(* CODESYS project WashingMachine (1).project

Project tree, tasks and I/O mapping:
  Device : CODESYS Control Win V3, 3S - Smart Software Solutions GmbH, version 3.5.15.10
    application Application
      libraries: Standard, * (System); VisuDialogs, * (System)
      task MainTask (cyclic, interval 100 ms, priority 1) calls Simulation_Program, GA_INSTANCES_prg, POLICY
      task VISU_TASK (cyclic, interval 100 ms, priority 31) calls VisuElems.Visu_Prg
      visualisation Visualization
      global variables GVL
      program Simulation_Program [ST]
      program BULLS_EYE_GA [SFC]: CHECK_DOOR_active, BUSY_active, LOCKING_DOOR_active, UNLOCKING_DOOR_active, END_active, END_exit, READY_active
      program TEMPERATURE_GA [SFC]: READY_active, BUSY_active, CHECK_TEMPERATURE_active, RESISTOR_ON_active, RESISTOR_OFF_active, CHECK_TEMPERATURE_exit
      program SOAP_GA [SFC]: CHECK_LEVEL_active, READY_active, BUSY_active, POURING_active, STOP_POURING_active, STOP_POURING_exit
      program WATER_GA [SFC]: READY_active, BUSY_active, FILLING_active, DRAINING_active, FILLING_exit, DRAINING_exit, END_active, END_exit, FAULT_OUT_DETECTOR_active, CHECK_LEVEL_active, FAULT_IN_DETECTOR_active
      program MOTOR_GA [SFC]: READY_active, BUSY_active, MOTOR_ON_active, MOTOR_OFF_active
      program POLICY [SFC]: RUN_PREWASH_exit, RUN_PREWASH_active, DOOR_UNLOCKED_active, CHECK_SOAP_active, RUN_PREWASH_NoRINSE_active, Init_exit, CHECK_DOOR_active, BULLS_EYE_LOCK_active, BULLS_EYE_LOCK_exit, RUN_WASH_active, RUN_WASH_exit, FINISHED_active, FAULT_MANAGER_active, Init_active, CHECK_TEMP_NUM_active, CHECK_PROG_NUM_active, BULLS_EYE_DOOR_UNLOCK_active, CHECK_STATE_active
      program PREWASH_WASH_POLICY [SFC]: Init_active, WATER_INTAKE_active, HEATING_active, FAULT_RESISTOR_active, EMPTYING_SOAP_active, MOTOR_ON_active, MOTOR_ON_exit, WATER_DRAIN_active, FAULT_OUT_VALVE_active, END_WASH_exit, END_WASH_active, HEATING_exit, EMPTYING_SOAP_exit, WATER_exit, RINSE_active, RINSE_exit, DUMMY_END_active, FAULT_HOT_DETECTOR_active, CHECK_FOR_STOP_active, WATER_DRAIN_entry
      program GA_INSTANCES_prg [FBD]
  text list GlobalTextList
*)

// Device/Application/GVL
{attribute 'qualified_only'}
VAR_GLOBAL
	temperature		: INT;		 	(*Sensor: current temperature of the water*)
	soaplevel		: INT; 			(*Sensor: current soap level*)
	waterlevel		: INT;			(*Sensor: current water level*)
	prog_number		: INT;			(*Input: program selected by the user*)
	temp_number		: INT; 			(*Input: temperature selected by the user*)
	run				: BOOL;			(*Input: if TRUE the washing machine works*)
	fillsoap		: BOOL; 		(*Input: if TRUE the soap tray is full*)
	bulls_eye_open	: BOOL := TRUE;	(*Input: if TRUE the door is open*)

	hot				: BOOL;			(*Actuator: if TRUE the resistor turns on*)
	motor_on		: BOOL;			(*Actuator: if TRUE the basket motor is turned on*)
	bulls_eye_lock	: BOOL;			(*Actuator: if TRUE the Door is locked*)
	emptysoap		: BOOL;			(*Actuator: if TRUE the soap tray is emptied*)
	fillwater		: BOOL;			(*Actuator: if TRUE the water is added*)
	emptywater		: BOOL;			(*Actuator: if TRUE the water is drained*)

	heat_alarm		: BOOL; 		(*Visualization: if TRUE alerts the user of the resistor fault*)
	water_in_alarm	: BOOL;			(*Visualization: if TRUE alerts the user of the water intake valve fault*)
	water_out_alarm	: BOOL; 		(*Visualization: if TRUE alerts the user of the water drain valve fault*)
	soap_alarm		: BOOL;			(*Visualization: if TRUE there is no soap*)
	prog_error		: BOOL;			(*Visualization: if TRUE the program selected is wrong*)
	temp_error		: BOOL;			(*Visualization: if TRUE the temperature selected is wrong*)
	rinse			: BOOL; 		(*Visualization: if TRUE the rinsing operation is going on*)
	prewash			: BOOL; 		(*Visualization: if TRUE the prewashing operation is going on*)
	wash			: BOOL; 		(*Visualization: if TRUE the washing operation is going on*)

	motor			: INT;			(*Only for simulation: angular position of the basket*)
	heat_fail		: BOOL;			(*Only for simulation: if TRUE the resistor cannot turn on*)
	water_in_fail	: BOOL;			(*Only for simulation: if TRUE the water intake valve is faulty*)
	water_out_fail	: BOOL;			(*Only for simulation: if TRUE the water drain valve is faulty*)
END_VAR

// Device/Application/Simulation_Program
PROGRAM Simulation_Program
VAR
		bulls_eye_open_past	:BOOL := TRUE;
END_VAR

(*Temperature value simulation*)
IF ((GVL.hot)AND(NOT GVL.heat_fail)) THEN 
	GVL.temperature := GVL.temperature + 1;
ELSE
	GVL.temperature := GVL.temperature - 1;
END_IF

IF GVL.temperature > 100 THEN 
	GVL.temperature := 100;
END_IF

IF GVL.temperature < 0 THEN 
	GVL.temperature := 0;
END_IF


(*Soap level simulation*)
IF GVL.fillsoap THEN 
	GVL.soaplevel := GVL.soaplevel + 5;
ELSIF GVL.emptysoap THEN 
	GVL.soaplevel := GVL.soaplevel - 3;
END_IF

IF GVL.soaplevel >= 50 THEN 
	GVL.soaplevel := 50;
	GVL.fillsoap := FALSE;
END_IF

IF GVL.soaplevel < 0 THEN 
	GVL.soaplevel := 0;
END_IF


(*Door state simulation*)
IF ((GVL.bulls_eye_open <> bulls_eye_open_past)AND(NOT GVL.bulls_eye_lock)) THEN 
	bulls_eye_open_past := GVL.bulls_eye_open ;
ELSIF GVL.bulls_eye_lock THEN
	GVL.bulls_eye_open := bulls_eye_open_past;
END_IF


(*Water level simulation*)
IF ((GVL.fillwater)AND(NOT GVL.water_in_fail)) THEN 
	GVL.waterlevel := GVL.waterlevel + 2;
ELSIF ((GVL.emptywater)AND(NOT GVL.water_out_fail)) THEN
	GVL.waterlevel := GVL.waterlevel - 4;
END_IF

IF GVL.waterlevel > 150 THEN 
	GVL.waterlevel := 150;
END_IF

IF GVL.waterlevel < 0 THEN 
	GVL.waterlevel := 0;
END_IF


(*Motor simulation*)
IF (GVL.motor_on) THEN 
	GVL.motor := GVL.motor + 10;
END_IF

IF GVL.motor > 360 THEN 
	GVL.motor := 0;
END_IF

END_PROGRAM

// Device/Application/GA_INSTANCES_prg
PROGRAM GA_INSTANCES_prg
VAR
END_VAR

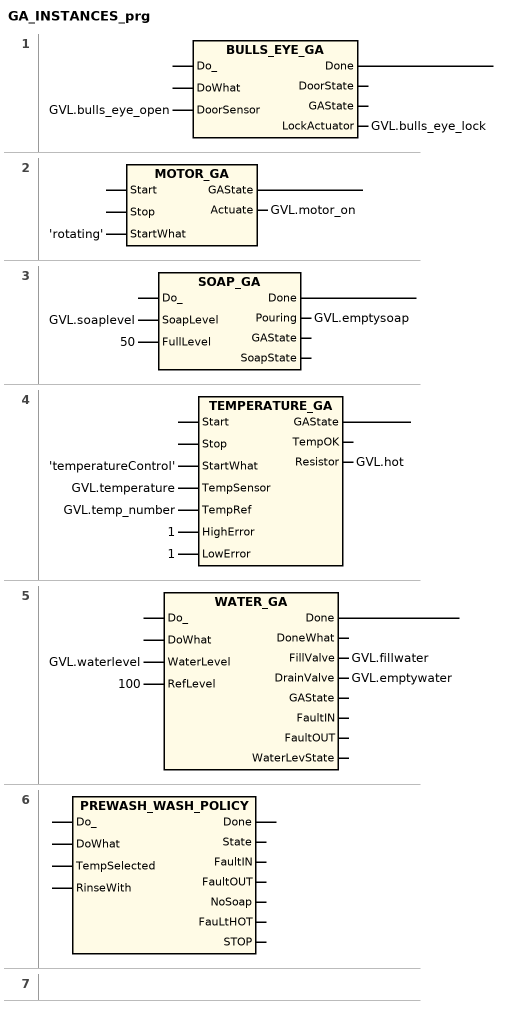
// NETWORK 1
BULLS_EYE_GA(DoorSensor := GVL.bulls_eye_open, LockActuator => GVL.bulls_eye_lock);

// NETWORK 2
MOTOR_GA(StartWhat := 'rotating', Actuate => GVL.motor_on);

// NETWORK 3
SOAP_GA(SoapLevel := GVL.soaplevel, FullLevel := 50, Pouring => GVL.emptysoap);

// NETWORK 4
TEMPERATURE_GA(StartWhat := 'temperatureControl', TempSensor := GVL.temperature, TempRef := GVL.temp_number, HighError := 1, LowError := 1, Resistor => GVL.hot);

// NETWORK 5
WATER_GA(WaterLevel := GVL.waterlevel, RefLevel := 100, FillValve => GVL.fillwater, DrainValve => GVL.emptywater);

// NETWORK 6
PREWASH_WASH_POLICY();

// NETWORK 7

END_PROGRAM

// Device/Application/BULLS_EYE_GA
PROGRAM BULLS_EYE_GA
//--------------------INPUT-----------------------
VAR_INPUT
	Do_:BOOL;
	DoWhat:STRING;
	DoorSensor:BOOL;
END_VAR
//-------------------OUTPUT-----------------------
VAR_OUTPUT
	Done:BOOL;
	DoorState:STRING;
	GAState:STRING;
	LockActuator:BOOL;
END_VAR
//--------------INTERNAL VARIABLES----------------
VAR
END_VAR

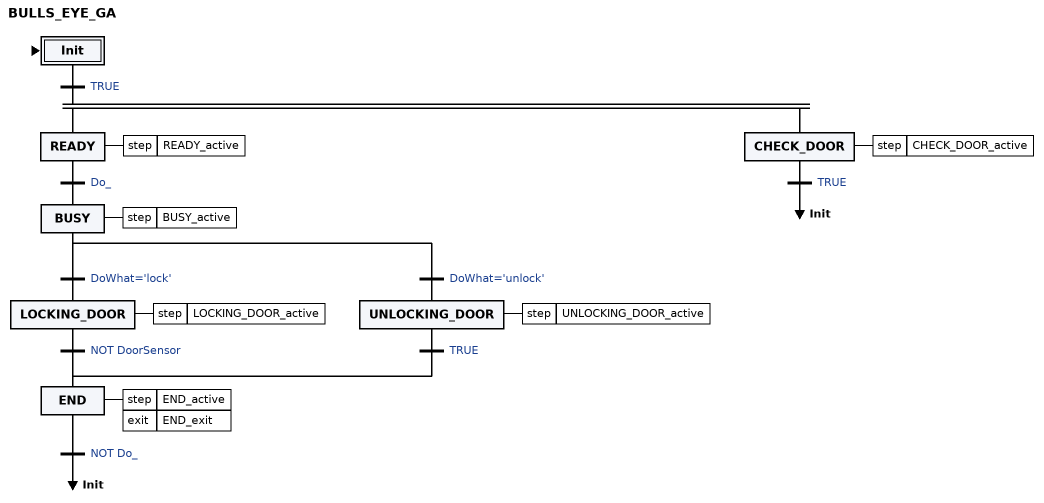
INITIAL_STEP Init:
END_STEP
TRANSITION FROM Init TO (READY, CHECK_DOOR)
    := TRUE;
END_TRANSITION
STEP READY:
    READY_active(N);  // step action
END_STEP
STEP CHECK_DOOR:
    CHECK_DOOR_active(N);  // step action
END_STEP
TRANSITION FROM CHECK_DOOR TO Init
    := TRUE;
END_TRANSITION
TRANSITION FROM READY TO BUSY
    := Do_;
END_TRANSITION
STEP BUSY:
    BUSY_active(N);  // step action
END_STEP
TRANSITION FROM BUSY TO LOCKING_DOOR
    := DoWhat='lock';
END_TRANSITION
STEP LOCKING_DOOR:
    LOCKING_DOOR_active(N);  // step action
END_STEP
TRANSITION FROM LOCKING_DOOR TO END
    := NOT DoorSensor;
END_TRANSITION
TRANSITION FROM BUSY TO UNLOCKING_DOOR
    := DoWhat='unlock';
END_TRANSITION
STEP UNLOCKING_DOOR:
    UNLOCKING_DOOR_active(N);  // step action
END_STEP
TRANSITION FROM UNLOCKING_DOOR TO END
    := TRUE;
END_TRANSITION
STEP END:
    END_active(N);  // step action
    END_exit(P0);  // exit action
END_STEP
TRANSITION FROM END TO Init
    := NOT Do_;
END_TRANSITION

ACTION CHECK_DOOR_active:
IF DoorSensor THEN
	DoorState:='open';
ELSE
	DoorState:='closed';
END_IF
END_ACTION

ACTION BUSY_active:
GAState:='busy';
END_ACTION

ACTION LOCKING_DOOR_active:
LockActuator:=TRUE;
END_ACTION

ACTION UNLOCKING_DOOR_active:
LockActuator:=FALSE;
END_ACTION

ACTION END_active:
Done:=TRUE;
END_ACTION

ACTION END_exit:
Done:=FALSE;
END_ACTION

ACTION READY_active:
GAState:='ready';
END_ACTION

END_PROGRAM

// Device/Application/MOTOR_GA
PROGRAM MOTOR_GA
//--------------------INPUT-----------------------
VAR_INPUT
	Start:BOOL;
	Stop:BOOL;
	StartWhat:STRING;
END_VAR
//-------------------OUTPUT-----------------------
VAR_OUTPUT
	GAState:STRING;
	Actuate:BOOL;
END_VAR
//--------------INTERNAL VARIABLES----------------
VAR
END_VAR

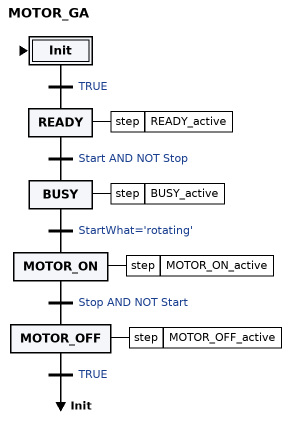
INITIAL_STEP Init:
END_STEP
TRANSITION FROM Init TO READY
    := TRUE;
END_TRANSITION
STEP READY:
    READY_active(N);  // step action
END_STEP
TRANSITION FROM READY TO BUSY
    := Start AND NOT Stop;
END_TRANSITION
STEP BUSY:
    BUSY_active(N);  // step action
END_STEP
TRANSITION FROM BUSY TO MOTOR_ON
    := StartWhat='rotating';
END_TRANSITION
STEP MOTOR_ON:
    MOTOR_ON_active(N);  // step action
END_STEP
TRANSITION FROM MOTOR_ON TO MOTOR_OFF
    := Stop AND NOT Start;
END_TRANSITION
STEP MOTOR_OFF:
    MOTOR_OFF_active(N);  // step action
END_STEP
TRANSITION FROM MOTOR_OFF TO Init
    := TRUE;
END_TRANSITION

ACTION READY_active:
GAState:='ready';
END_ACTION

ACTION BUSY_active:
GAState:='busy';
END_ACTION

ACTION MOTOR_ON_active:
Actuate:=TRUE;
END_ACTION

ACTION MOTOR_OFF_active:
Actuate:=FALSE;
END_ACTION

END_PROGRAM

// Device/Application/SOAP_GA
PROGRAM SOAP_GA
//--------------------INPUT-----------------------
VAR_INPUT
	Do_:BOOL;
	SoapLevel:INT;
	FullLevel:INT;
END_VAR
//-------------------OUTPUT-----------------------
VAR_OUTPUT
	Done:BOOL;
	Pouring:BOOL;
	GAState:STRING;
	SoapState:STRING;
END_VAR
//--------------INTERNAL VARIABLES----------------
VAR
	PouringTime:TIME := T#10S;
END_VAR

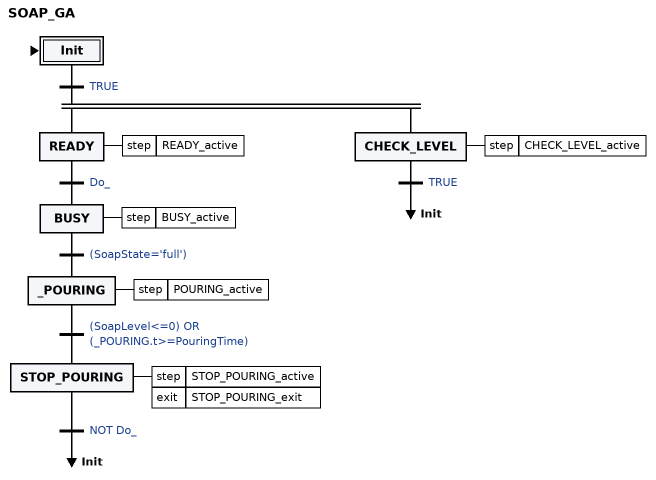
INITIAL_STEP Init:
END_STEP
TRANSITION FROM Init TO (READY, CHECK_LEVEL)
    := TRUE;
END_TRANSITION
STEP READY:
    READY_active(N);  // step action
END_STEP
STEP CHECK_LEVEL:
    CHECK_LEVEL_active(N);  // step action
END_STEP
TRANSITION FROM CHECK_LEVEL TO Init
    := TRUE;
END_TRANSITION
TRANSITION FROM READY TO BUSY
    := Do_;
END_TRANSITION
STEP BUSY:
    BUSY_active(N);  // step action
END_STEP
TRANSITION FROM BUSY TO _POURING
    := (SoapState='full');
END_TRANSITION
STEP _POURING:
    POURING_active(N);  // step action
END_STEP
TRANSITION FROM _POURING TO STOP_POURING
    := (SoapLevel<=0) OR (_POURING.t>=PouringTime);
END_TRANSITION
STEP STOP_POURING:
    STOP_POURING_active(N);  // step action
    STOP_POURING_exit(P0);  // exit action
END_STEP
TRANSITION FROM STOP_POURING TO Init
    := NOT Do_;
END_TRANSITION

ACTION CHECK_LEVEL_active:
IF SoapLevel>=FullLevel THEN
	SoapState:='full';
ELSE 
	SoapState:='notfull';	
END_IF
END_ACTION

ACTION READY_active:
GAState:='ready';
END_ACTION

ACTION BUSY_active:
GAState:='busy';
END_ACTION

ACTION POURING_active:
Pouring:=TRUE;
END_ACTION

ACTION STOP_POURING_active:
Pouring:=FALSE;
Done:=TRUE;
END_ACTION

ACTION STOP_POURING_exit:
Done:=FALSE;
END_ACTION

END_PROGRAM

// Device/Application/TEMPERATURE_GA
PROGRAM TEMPERATURE_GA
//--------------------INPUT-----------------------
VAR_INPUT
	Start:BOOL;
	Stop:BOOL;
	StartWhat:STRING;
	TempSensor:INT;
	TempRef:INT;
	HighError:INT;
	LowError:INT;
END_VAR
//-------------------OUTPUT-----------------------
VAR_OUTPUT
	GAState:STRING;
	TempOK:BOOL;
	Resistor:BOOL;
END_VAR
//--------------INTERNAL VARIABLES----------------
VAR
END_VAR

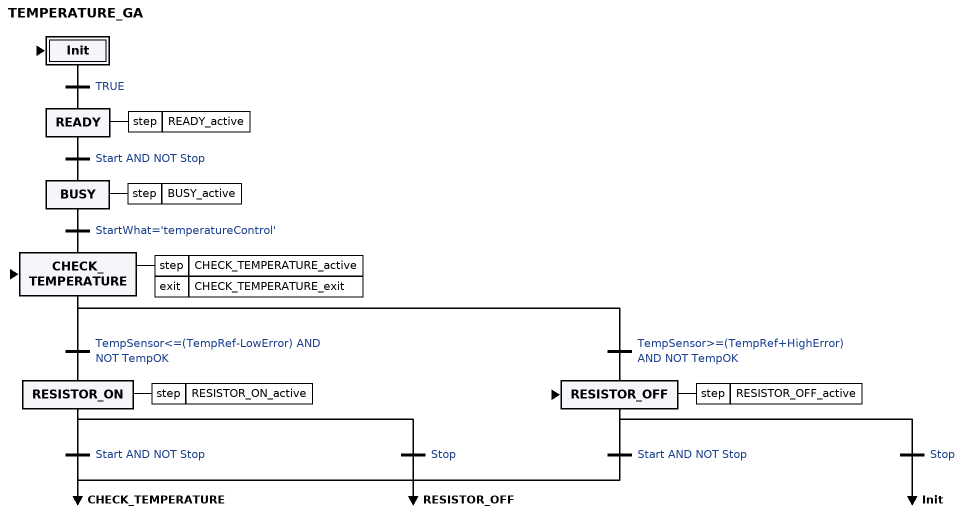
INITIAL_STEP Init:
END_STEP
TRANSITION FROM Init TO READY
    := TRUE;
END_TRANSITION
STEP READY:
    READY_active(N);  // step action
END_STEP
TRANSITION FROM READY TO BUSY
    := Start AND NOT Stop;
END_TRANSITION
STEP BUSY:
    BUSY_active(N);  // step action
END_STEP
TRANSITION FROM BUSY TO CHECK_TEMPERATURE
    := StartWhat='temperatureControl';
END_TRANSITION
STEP CHECK_TEMPERATURE:
    CHECK_TEMPERATURE_active(N);  // step action
    CHECK_TEMPERATURE_exit(P0);  // exit action
END_STEP
TRANSITION FROM CHECK_TEMPERATURE TO RESISTOR_ON
    := TempSensor<=(TempRef-LowError) AND NOT TempOK;
END_TRANSITION
STEP RESISTOR_ON:
    RESISTOR_ON_active(N);  // step action
END_STEP
TRANSITION FROM RESISTOR_ON TO CHECK_TEMPERATURE
    := Start AND NOT Stop;
END_TRANSITION
TRANSITION FROM RESISTOR_ON TO RESISTOR_OFF
    := Stop;
END_TRANSITION
TRANSITION FROM CHECK_TEMPERATURE TO RESISTOR_OFF
    := TempSensor>=(TempRef+HighError) AND NOT TempOK;
END_TRANSITION
STEP RESISTOR_OFF:
    RESISTOR_OFF_active(N);  // step action
END_STEP
TRANSITION FROM RESISTOR_OFF TO CHECK_TEMPERATURE
    := Start AND NOT Stop;
END_TRANSITION
TRANSITION FROM RESISTOR_OFF TO Init
    := Stop;
END_TRANSITION

ACTION READY_active:
GAState:='ready';
TempOK:=FALSE;
END_ACTION

ACTION BUSY_active:
GAState:='busy';
END_ACTION

ACTION CHECK_TEMPERATURE_active:
IF (TempSensor <= (TempRef + HighError)) AND (TempSensor >= (TempRef - LowError)) THEN
	TempOK:=TRUE;
ELSE
	TempOK:=FALSE;
END_IF
END_ACTION

ACTION RESISTOR_ON_active:
Resistor:=TRUE;
END_ACTION

ACTION RESISTOR_OFF_active:
Resistor:=FALSE;
END_ACTION

ACTION CHECK_TEMPERATURE_exit:
TempOK:=FALSE;
END_ACTION

END_PROGRAM

// Device/Application/WATER_GA
PROGRAM WATER_GA
//--------------------INPUT-----------------------
VAR_INPUT
	Do_:BOOL;
	DoWhat:STRING;
	WaterLevel:INT;
	RefLevel:INT;
END_VAR
//-------------------OUTPUT-----------------------
VAR_OUTPUT
	Done:BOOL;
	DoneWhat:STRING;
	FillValve:BOOL;
	DrainValve:BOOL;
	GAState:STRING;
	FaultIN:BOOL;
	FaultOUT:BOOL;
	WaterLevState:STRING;
END_VAR
//--------------INTERNAL VARIABLES----------------
VAR
	TimeFilling:TIME :=T#10S;
	TimeDraining:TIME :=T#10S;
    PrevLev:INT:=0;
	Count:INT:=0;
END_VAR

//WaterLevel>=RefLevel OR FILLING.t>TimeFilling
//WaterLevel<=0 OR DRAINING.t>TimeDraining

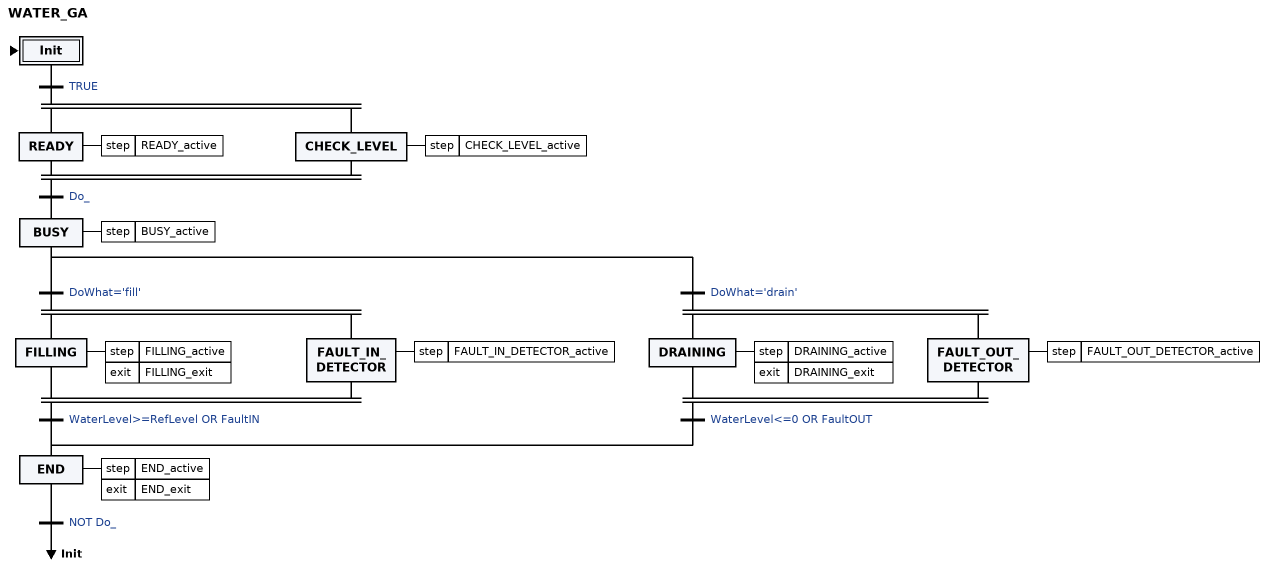
INITIAL_STEP Init:
END_STEP
TRANSITION FROM Init TO (READY, CHECK_LEVEL)
    := TRUE;
END_TRANSITION
STEP READY:
    READY_active(N);  // step action
END_STEP
STEP CHECK_LEVEL:
    CHECK_LEVEL_active(N);  // step action
END_STEP
TRANSITION FROM (READY, CHECK_LEVEL) TO BUSY
    := Do_;
END_TRANSITION
STEP BUSY:
    BUSY_active(N);  // step action
END_STEP
TRANSITION FROM BUSY TO (FILLING, FAULT_IN_DETECTOR)
    := DoWhat='fill';
END_TRANSITION
STEP FILLING:
    FILLING_active(N);  // step action
    FILLING_exit(P0);  // exit action
END_STEP
STEP FAULT_IN_DETECTOR:
    FAULT_IN_DETECTOR_active(N);  // step action
END_STEP
TRANSITION FROM (FILLING, FAULT_IN_DETECTOR) TO END
    := WaterLevel>=RefLevel OR FaultIN;
END_TRANSITION
TRANSITION FROM BUSY TO (DRAINING, FAULT_OUT_DETECTOR)
    := DoWhat='drain';
END_TRANSITION
STEP DRAINING:
    DRAINING_active(N);  // step action
    DRAINING_exit(P0);  // exit action
END_STEP
STEP FAULT_OUT_DETECTOR:
    FAULT_OUT_DETECTOR_active(N);  // step action
END_STEP
TRANSITION FROM (DRAINING, FAULT_OUT_DETECTOR) TO END
    := WaterLevel<=0 OR FaultOUT;
END_TRANSITION
STEP END:
    END_active(N);  // step action
    END_exit(P0);  // exit action
END_STEP
TRANSITION FROM END TO Init
    := NOT Do_;
END_TRANSITION

ACTION READY_active:
GAState:='ready';
END_ACTION

ACTION BUSY_active:
GAState:='busy';
END_ACTION

ACTION FILLING_active:
IF WaterLevel<RefLevel THEN
	WaterLevState:='notfull';	
	FillValve:=TRUE;
	DrainValve:=FALSE;
ELSE
WaterLevState:='full';	
END_IF
END_ACTION

ACTION DRAINING_active:
IF WaterLevel>0THEN
	WaterLevState:='full';	
	FillValve:=FALSE;
	DrainValve:=TRUE;
ELSE
	WaterLevState:='notfull';	
END_IF
END_ACTION

ACTION FILLING_exit:
FillValve:=FALSE;
DoneWhat:='fill';
END_ACTION

ACTION DRAINING_exit:
DrainValve:=FALSE;
DoneWhat:='drain';
END_ACTION

ACTION END_active:
Done:=TRUE;
PrevLev:=0;
END_ACTION

ACTION END_exit:
Done:=FALSE;
Count:=0;
END_ACTION

ACTION FAULT_OUT_DETECTOR_active:
//fault detection in the water_in_valve

FaultOUT:=FALSE;
IF Count=0THEN
	PrevLev:=WaterLevel;
END_IF
Count:=Count+1;
IF Count=20 THEN
	IF PrevLev <= WaterLevel THEN
		FaultOUT:=TRUE;
	ELSE
		FaultOUT:=FALSE;
	END_IF
	Count:=0;
END_IF
END_ACTION

ACTION CHECK_LEVEL_active:
IF WaterLevel>=RefLevel THEN
	WaterLevState:='full';
ELSE 
	WaterLevState:='notfull';	
END_IF

FaultIN:=FALSE;
FaultOUT:=FALSE;
END_ACTION

ACTION FAULT_IN_DETECTOR_active:
//fault detection in the water_in_valve

FaultIN:=FALSE;
Count:=Count+1;
IF Count=20 THEN
	IF PrevLev >= WaterLevel THEN
		FaultIN:=TRUE;
	ELSE
		FaultIN:=FALSE;
	END_IF
	PrevLev:=WaterLevel;
	Count:=0;
END_IF
END_ACTION

END_PROGRAM

// Device/Application/PREWASH_WASH_POLICY
PROGRAM PREWASH_WASH_POLICY
//--------------------INPUT-----------------------
VAR_INPUT
	Do_:BOOL;
	DoWhat:STRING;
	TempSelected:INT;
	RinseWith:BOOL;
END_VAR
//-------------------OUTPUT-----------------------
VAR_OUTPUT
	Done:BOOL;
	State:STRING;
	FaultIN:BOOL;
	FaultOUT:BOOL;
	NoSoap:BOOL;
	FauLtHOT:BOOL;
	STOP:BOOL;
END_VAR
//--------------INTERNAL VARIABLES----------------
VAR
	OK:BOOL;
	HeatingMaxTime:TIME:=T#10S;
	SoapOK:BOOL;
	Count:INT:=0;
	PrevTemp:INT:=0;
END_VAR

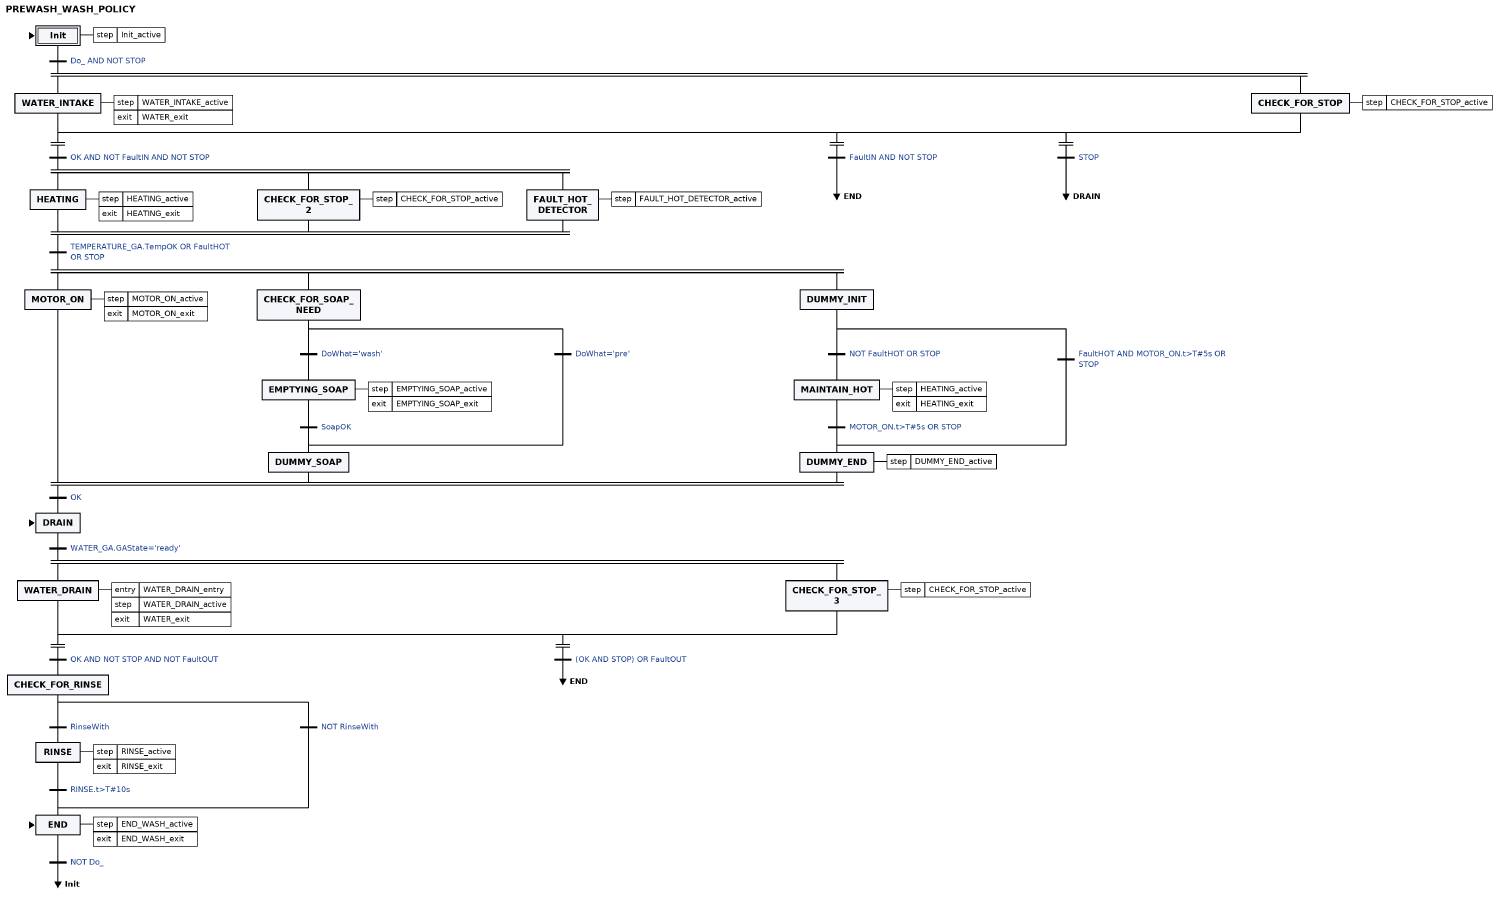
INITIAL_STEP Init:
    Init_active(N);  // step action
END_STEP
TRANSITION FROM Init TO (WATER_INTAKE, CHECK_FOR_STOP)
    := Do_ AND NOT STOP;
END_TRANSITION
STEP WATER_INTAKE:
    WATER_INTAKE_active(N);  // step action
    WATER_exit(P0);  // exit action
END_STEP
STEP CHECK_FOR_STOP:
    CHECK_FOR_STOP_active(N);  // step action
END_STEP
TRANSITION FROM (WATER_INTAKE, CHECK_FOR_STOP) TO (HEATING, CHECK_FOR_STOP_2, FAULT_HOT_DETECTOR)
    := OK AND NOT FaultIN AND NOT STOP;
END_TRANSITION
TRANSITION FROM (WATER_INTAKE, CHECK_FOR_STOP) TO END
    := FaultIN AND NOT STOP;
END_TRANSITION
TRANSITION FROM (WATER_INTAKE, CHECK_FOR_STOP) TO DRAIN
    := STOP;
END_TRANSITION
STEP HEATING:
    HEATING_active(N);  // step action
    HEATING_exit(P0);  // exit action
END_STEP
STEP CHECK_FOR_STOP_2:
    CHECK_FOR_STOP_active(N);  // step action
END_STEP
STEP FAULT_HOT_DETECTOR:
    FAULT_HOT_DETECTOR_active(N);  // step action
END_STEP
TRANSITION FROM (HEATING, CHECK_FOR_STOP_2, FAULT_HOT_DETECTOR) TO (MOTOR_ON, CHECK_FOR_SOAP_NEED, DUMMY_INIT)
    := TEMPERATURE_GA.TempOK OR FaultHOT OR STOP;
END_TRANSITION
STEP MOTOR_ON:
    MOTOR_ON_active(N);  // step action
    MOTOR_ON_exit(P0);  // exit action
END_STEP
STEP CHECK_FOR_SOAP_NEED:
END_STEP
TRANSITION FROM CHECK_FOR_SOAP_NEED TO EMPTYING_SOAP
    := DoWhat='wash';
END_TRANSITION
STEP EMPTYING_SOAP:
    EMPTYING_SOAP_active(N);  // step action
    EMPTYING_SOAP_exit(P0);  // exit action
END_STEP
TRANSITION FROM EMPTYING_SOAP TO DUMMY_SOAP
    := SoapOK;
END_TRANSITION
TRANSITION FROM CHECK_FOR_SOAP_NEED TO DUMMY_SOAP
    := DoWhat='pre';
END_TRANSITION
STEP DUMMY_SOAP:
END_STEP
STEP DUMMY_INIT:
END_STEP
TRANSITION FROM DUMMY_INIT TO MAINTAIN_HOT
    := NOT FaultHOT OR STOP;
END_TRANSITION
STEP MAINTAIN_HOT:
    HEATING_active(N);  // step action
    HEATING_exit(P0);  // exit action
END_STEP
TRANSITION FROM MAINTAIN_HOT TO DUMMY_END
    := MOTOR_ON.t>T#5s OR STOP;
END_TRANSITION
TRANSITION FROM DUMMY_INIT TO DUMMY_END
    := FaultHOT AND MOTOR_ON.t>T#5s OR STOP;
END_TRANSITION
STEP DUMMY_END:
    DUMMY_END_active(N);  // step action
END_STEP
TRANSITION FROM (MOTOR_ON, DUMMY_SOAP, DUMMY_END) TO DRAIN
    := OK;
END_TRANSITION
STEP DRAIN:
END_STEP
TRANSITION FROM DRAIN TO (WATER_DRAIN, CHECK_FOR_STOP_3)
    := WATER_GA.GAState='ready';
END_TRANSITION
STEP WATER_DRAIN:
    WATER_DRAIN_entry(P1);  // entry action
    WATER_DRAIN_active(N);  // step action
    WATER_exit(P0);  // exit action
END_STEP
STEP CHECK_FOR_STOP_3:
    CHECK_FOR_STOP_active(N);  // step action
END_STEP
TRANSITION FROM (WATER_DRAIN, CHECK_FOR_STOP_3) TO CHECK_FOR_RINSE
    := OK AND NOT STOP AND NOT FaultOUT;
END_TRANSITION
TRANSITION FROM (WATER_DRAIN, CHECK_FOR_STOP_3) TO END
    := (OK AND STOP) OR FaultOUT;
END_TRANSITION
STEP CHECK_FOR_RINSE:
END_STEP
TRANSITION FROM CHECK_FOR_RINSE TO RINSE
    := RinseWith;
END_TRANSITION
STEP RINSE:
    RINSE_active(N);  // step action
    RINSE_exit(P0);  // exit action
END_STEP
TRANSITION FROM RINSE TO END
    := RINSE.t>T#10s;
END_TRANSITION
TRANSITION FROM CHECK_FOR_RINSE TO END
    := NOT RinseWith;
END_TRANSITION
STEP END:
    END_WASH_active(N);  // step action
    END_WASH_exit(P0);  // exit action
END_STEP
TRANSITION FROM END TO Init
    := NOT Do_;
END_TRANSITION

ACTION Init_active:
State:='init';
FaultIN:=FALSE;
FaultOUT:=FALSE;
NoSoap:=FALSE;
FauLtHOT:=FALSE;
IF GVL.run THEN
	STOP:=FALSE;
ELSE
	STOP:=TRUE;
END_IF
END_ACTION

ACTION WATER_INTAKE_active:
FaultIN:=FALSE;
IF WATER_GA.WaterLevState='notfull' THEN

		IF WATER_GA.GAState='ready' THEN
			WATER_GA.Do_:=TRUE;
			WATER_GA.DoWhat:='fill';
		END_IF

		IF WATER_GA.Done AND WATER_GA.GAState='busy' THEN
			FaultIN:=WATER_GA.FaultIN;
			OK:=TRUE;
		END_IF
		
	ELSE
		OK:=TRUE;
END_IF	
IF NOT(State='fault') THEN
	State:=DoWhat;
END_IF
END_ACTION

ACTION HEATING_active:
FaultHOT:=FALSE;
IF TEMPERATURE_GA.GAState= 'ready' THEN
		TEMPERATURE_GA.Start:=TRUE;
		TEMPERATURE_GA.Stop:=FALSE;
END_IF
END_ACTION

ACTION FAULT_RESISTOR_active:
FaultHOT:=TRUE;
State:='fault';
END_ACTION

ACTION EMPTYING_SOAP_active:
NoSoap:=FALSE;
IF SOAP_GA.SoapState='full' THEN
	NoSoap:=FALSE;
ELSE
	NoSoap:=TRUE;
END_IF

IF SOAP_GA.SoapLevel>0 THEN
	IF SOAP_GA.GAState='ready'THEN
		SOAP_GA.Do_:=TRUE;
	END_IF
	IF SOAP_GA.Done AND SOAP_GA.GAState='busy' THEN
		SOAP_GA.Do_:=FALSE;
		SoapOK:=SOAP_GA.Done;
	END_IF
ELSE
	SoapOK:=TRUE;
END_IF
END_ACTION

ACTION MOTOR_ON_active:
IF MOTOR_GA.GAState= 'ready' THEN
		MOTOR_GA.Start:=TRUE;
		MOTOR_GA.Stop:=FALSE;
END_IF
END_ACTION

ACTION MOTOR_ON_exit:
IF MOTOR_GA.GAState= 'busy' THEN
		MOTOR_GA.Start:=FALSE;
		MOTOR_GA.Stop:=TRUE;
END_IF
END_ACTION

ACTION WATER_DRAIN_active:
FaultOUT:=FALSE;
IF WATER_GA.WaterLevState='full'THEN
		
		IF WATER_GA.GAState='ready' THEN
			WATER_GA.Do_:=TRUE;
			WATER_GA.DoWhat:='drain';
		END_IF

		IF WATER_GA.Done AND WATER_GA.GAState='busy' THEN
			FaultOUT:=WATER_GA.FaultOUT;
			OK:=TRUE;
		END_IF
		
	ELSE
		OK:=TRUE;
END_IF
END_ACTION

ACTION FAULT_OUT_VALVE_active:
GVL.water_out_alarm:=TRUE;
FaultOUT:=TRUE;
END_ACTION

ACTION END_WASH_exit:
Done:=FALSE;
State:='init';
STOP:=FALSE;
END_ACTION

ACTION END_WASH_active:
IF ((NOT FaultIN) AND (NOT FaultOUT) AND (NOT FaultHOT))THEN
	State:='end';
ELSE
	State:='fault';
END_IF

IF GVL.run THEN
	STOP:=FALSE;
ELSE
	STOP:=TRUE;
END_IF

Done:=TRUE;
Count:=0;
PrevTemp:=0;
END_ACTION

ACTION HEATING_exit:
IF TEMPERATURE_GA.GAState= 'busy' THEN
		TEMPERATURE_GA.Start:=FALSE;
		TEMPERATURE_GA.Stop:=TRUE;
END_IF
Count:=0;
STOP:=FALSE;
END_ACTION

ACTION EMPTYING_SOAP_exit:
SoapOK:=FALSE;
END_ACTION

ACTION WATER_exit:
OK:=FALSE;
WATER_GA.Do_:=FALSE;
STOP:=FALSE;
END_ACTION

ACTION RINSE_active:
IF MOTOR_GA.GAState= 'ready' THEN
		MOTOR_GA.Start:=TRUE;
		MOTOR_GA.Stop:=FALSE;
END_IF
IF NOT(State='fault') THEN
	State:='rinse';
END_IF
END_ACTION

ACTION RINSE_exit:
IF MOTOR_GA.GAState= 'busy' THEN
		MOTOR_GA.Start:=FALSE;
		MOTOR_GA.Stop:=TRUE;
END_IF
END_ACTION

ACTION DUMMY_END_active:
OK:=TRUE;
END_ACTION

ACTION FAULT_HOT_DETECTOR_active:
FaultHOT:=FALSE;
Count:=Count+1;
IF Count=20 THEN
	IF PrevTemp >= TEMPERATURE_GA.TempSensor THEN
		FaultHOT:=TRUE;
		State:='fault';
	ELSE
		FaultHOT:=FALSE;
	END_IF
	PrevTemp:=TEMPERATURE_GA.TempSensor;
	Count:=0;
END_IF
END_ACTION

ACTION CHECK_FOR_STOP_active:
IF GVL.run THEN
	STOP:=FALSE;
ELSE
	STOP:=TRUE;
END_IF
END_ACTION

ACTION WATER_DRAIN_entry:
OK:=FALSE;
END_ACTION

END_PROGRAM

// Device/Application/POLICY
PROGRAM POLICY
VAR
	TempNumOK:BOOL;
	ProgNumOK:BOOL;
	RunOK:BOOL;
	WashOK:BOOL;
	STOP:BOOL;
	DoorOK:BOOL;
	TempOK:BOOL;


END_VAR

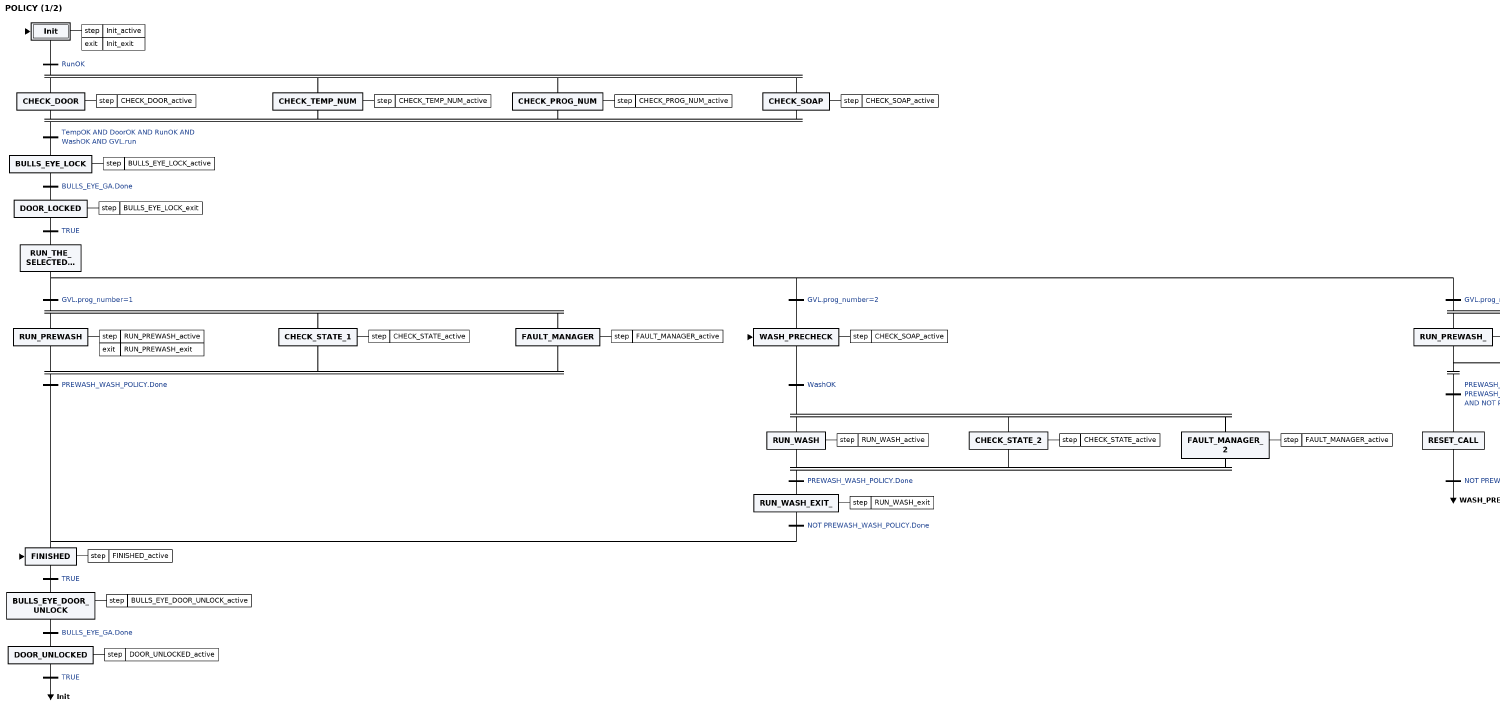
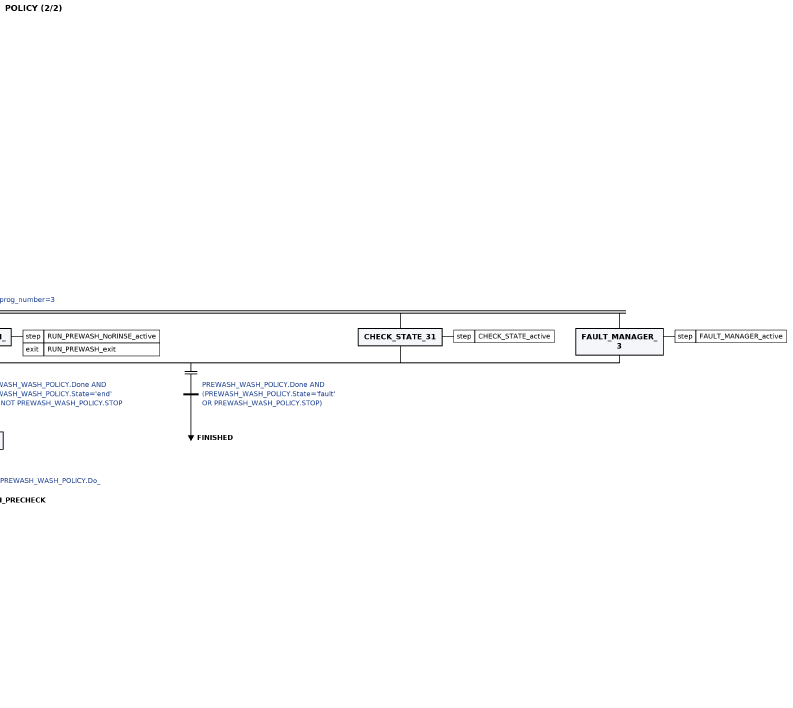
INITIAL_STEP Init:
    Init_active(N);  // step action
    Init_exit(P0);  // exit action
END_STEP
TRANSITION FROM Init TO (CHECK_DOOR, CHECK_TEMP_NUM, CHECK_PROG_NUM, CHECK_SOAP)
    := RunOK;
END_TRANSITION
STEP CHECK_DOOR:
    CHECK_DOOR_active(N);  // step action
END_STEP
STEP CHECK_TEMP_NUM:
    CHECK_TEMP_NUM_active(N);  // step action
END_STEP
STEP CHECK_PROG_NUM:
    CHECK_PROG_NUM_active(N);  // step action
END_STEP
STEP CHECK_SOAP:
    CHECK_SOAP_active(N);  // step action
END_STEP
TRANSITION FROM (CHECK_DOOR, CHECK_TEMP_NUM, CHECK_PROG_NUM, CHECK_SOAP) TO BULLS_EYE_LOCK
    := TempOK AND DoorOK AND RunOK AND WashOK AND GVL.run;
END_TRANSITION
STEP BULLS_EYE_LOCK:
    BULLS_EYE_LOCK_active(N);  // step action
END_STEP
TRANSITION FROM BULLS_EYE_LOCK TO DOOR_LOCKED
    := BULLS_EYE_GA.Done;
END_TRANSITION
STEP DOOR_LOCKED:
    BULLS_EYE_LOCK_exit(N);  // step action
END_STEP
TRANSITION FROM DOOR_LOCKED TO RUN_THE_SELECTED_PROGRAM
    := TRUE;
END_TRANSITION
STEP RUN_THE_SELECTED_PROGRAM:
END_STEP
TRANSITION FROM RUN_THE_SELECTED_PROGRAM TO (RUN_PREWASH, CHECK_STATE_1, FAULT_MANAGER)
    := GVL.prog_number=1;
END_TRANSITION
STEP RUN_PREWASH:
    RUN_PREWASH_active(N);  // step action
    RUN_PREWASH_exit(P0);  // exit action
END_STEP
STEP CHECK_STATE_1:
    CHECK_STATE_active(N);  // step action
END_STEP
STEP FAULT_MANAGER:
    FAULT_MANAGER_active(N);  // step action
END_STEP
TRANSITION FROM (RUN_PREWASH, CHECK_STATE_1, FAULT_MANAGER) TO FINISHED
    := PREWASH_WASH_POLICY.Done;
END_TRANSITION
TRANSITION FROM RUN_THE_SELECTED_PROGRAM TO WASH_PRECHECK
    := GVL.prog_number=2;
END_TRANSITION
STEP WASH_PRECHECK:
    CHECK_SOAP_active(N);  // step action
END_STEP
TRANSITION FROM WASH_PRECHECK TO (RUN_WASH, CHECK_STATE_2, FAULT_MANAGER_2)
    := WashOK;
END_TRANSITION
STEP RUN_WASH:
    RUN_WASH_active(N);  // step action
END_STEP
STEP CHECK_STATE_2:
    CHECK_STATE_active(N);  // step action
END_STEP
STEP FAULT_MANAGER_2:
    FAULT_MANAGER_active(N);  // step action
END_STEP
TRANSITION FROM (RUN_WASH, CHECK_STATE_2, FAULT_MANAGER_2) TO RUN_WASH_EXIT_
    := PREWASH_WASH_POLICY.Done;
END_TRANSITION
STEP RUN_WASH_EXIT_:
    RUN_WASH_exit(N);  // step action
END_STEP
TRANSITION FROM RUN_WASH_EXIT_ TO FINISHED
    := NOT PREWASH_WASH_POLICY.Done;
END_TRANSITION
TRANSITION FROM RUN_THE_SELECTED_PROGRAM TO (RUN_PREWASH_, CHECK_STATE_31, FAULT_MANAGER_3)
    := GVL.prog_number=3;
END_TRANSITION
STEP RUN_PREWASH_:
    RUN_PREWASH_NoRINSE_active(N);  // step action
    RUN_PREWASH_exit(P0);  // exit action
END_STEP
STEP CHECK_STATE_31:
    CHECK_STATE_active(N);  // step action
END_STEP
STEP FAULT_MANAGER_3:
    FAULT_MANAGER_active(N);  // step action
END_STEP
TRANSITION FROM (RUN_PREWASH_, CHECK_STATE_31, FAULT_MANAGER_3) TO RESET_CALL
    := PREWASH_WASH_POLICY.Done AND PREWASH_WASH_POLICY.State='end' AND NOT PREWASH_WASH_POLICY.STOP;
END_TRANSITION
STEP RESET_CALL:
END_STEP
TRANSITION FROM RESET_CALL TO WASH_PRECHECK
    := NOT PREWASH_WASH_POLICY.Do_;
END_TRANSITION
TRANSITION FROM (RUN_PREWASH_, CHECK_STATE_31, FAULT_MANAGER_3) TO FINISHED
    := PREWASH_WASH_POLICY.Done AND (PREWASH_WASH_POLICY.State='fault' OR PREWASH_WASH_POLICY.STOP);
END_TRANSITION
STEP FINISHED:
    FINISHED_active(N);  // step action
END_STEP
TRANSITION FROM FINISHED TO BULLS_EYE_DOOR_UNLOCK
    := TRUE;
END_TRANSITION
STEP BULLS_EYE_DOOR_UNLOCK:
    BULLS_EYE_DOOR_UNLOCK_active(N);  // step action
END_STEP
TRANSITION FROM BULLS_EYE_DOOR_UNLOCK TO DOOR_UNLOCKED
    := BULLS_EYE_GA.Done;
END_TRANSITION
STEP DOOR_UNLOCKED:
    DOOR_UNLOCKED_active(N);  // step action
END_STEP
TRANSITION FROM DOOR_UNLOCKED TO Init
    := TRUE;
END_TRANSITION

ACTION RUN_PREWASH_exit:
PREWASH_WASH_POLICY.Do_:=FALSE;
END_ACTION

ACTION RUN_PREWASH_active:
PREWASH_WASH_POLICY.Do_:=TRUE;
PREWASH_WASH_POLICY.DoWhat:='pre';
PREWASH_WASH_POLICY.RinseWith:=TRUE;
END_ACTION

ACTION DOOR_UNLOCKED_active:
IF BULLS_EYE_GA.GAState='busy' THEN
	BULLS_EYE_GA.Do_:=FALSE;
END_IF
END_ACTION

ACTION CHECK_SOAP_active:
IF (SOAP_GA.SoapState='full')OR(GVL.prog_number=1)THEN
	WashOK:=TRUE;
	GVL.soap_alarm:=FALSE;
ELSE
	WashOK:=FALSE;
	GVL.soap_alarm:=TRUE;
END_IF
END_ACTION

ACTION RUN_PREWASH_NoRINSE_active:
PREWASH_WASH_POLICY.Do_:=TRUE;
PREWASH_WASH_POLICY.DoWhat:='pre';
PREWASH_WASH_POLICY.RinseWith:=FALSE;
END_ACTION

ACTION Init_exit:
RunOK:=FALSE;
END_ACTION

ACTION CHECK_DOOR_active:
IF BULLS_EYE_GA.DoorState='open'THEN
	DoorOK:=FALSE;
END_IF

IF BULLS_EYE_GA.DoorState='closed' THEN
	DoorOK:=TRUE;
END_IF
END_ACTION

ACTION BULLS_EYE_LOCK_active:
IF BULLS_EYE_GA.GAState='ready' THEN
	BULLS_EYE_GA.Do_:=TRUE;
	BULLS_EYE_GA.DoWhat:='lock';
END_IF
END_ACTION

ACTION BULLS_EYE_LOCK_exit:
IF BULLS_EYE_GA.GAState='busy' THEN
	BULLS_EYE_GA.Do_:=FALSE;
END_IF
END_ACTION

ACTION RUN_WASH_active:
PREWASH_WASH_POLICY.Do_:=TRUE;
PREWASH_WASH_POLICY.DoWhat:='wash';
PREWASH_WASH_POLICY.RinseWith:=TRUE;
END_ACTION

ACTION RUN_WASH_exit:
PREWASH_WASH_POLICY.Do_:=FALSE;
END_ACTION

ACTION FINISHED_active:
GVL.run:=FALSE;
END_ACTION

ACTION FAULT_MANAGER_active:
IF PREWASH_WASH_POLICY.FaultIN THEN
	GVL.water_in_alarm:=TRUE;
ELSE
	GVL.water_in_alarm:=STOP:=FALSE;
END_IF
IF PREWASH_WASH_POLICY.FaultOUT THEN
	GVL.water_out_alarm:=TRUE;
ELSE
	GVL.water_OUT_alarm:=STOP:=FALSE;
END_IF
IF PREWASH_WASH_POLICY.FaultHOT THEN
	GVL.heat_alarm:=TRUE;
ELSE
	GVL.heat_alarm:=FALSE;
END_IF
IF PREWASH_WASH_POLICY.NoSoap THEN
	GVL.soap_alarm:=TRUE;
	WashOK:=FALSE;
ELSE
	GVL.soap_alarm:=FALSE;
	WashOK:=TRUE;
END_IF
END_ACTION

ACTION Init_active:
IF GVL.water_in_alarm OR GVL.water_out_alarm THEN
	RunOK:=FALSE;
ELSE
	RunOK:=TRUE;
END_IF
END_ACTION

ACTION CHECK_TEMP_NUM_active:
IF (GVL.temp_number=30)OR(GVL.temp_number=60)OR(GVL.temp_number=90)THEN
	TempOK:=TRUE;
	GVL.temp_error:=FALSE;
ELSE
	TempOK:=FALSE;
	GVL.temp_error:=TRUE;
END_IF
END_ACTION

ACTION CHECK_PROG_NUM_active:
IF (GVL.prog_number=1) OR (GVL.prog_number=2) OR (GVL.prog_number=3) THEN
	RunOK:=TRUE;
	GVL.prog_error:=FALSE;
ELSE
	RunOK:=FALSE;
	GVL.prog_error:=TRUE;
END_IF
END_ACTION

ACTION BULLS_EYE_DOOR_UNLOCK_active:
IF BULLS_EYE_GA.GAState='ready' THEN
	BULLS_EYE_GA.Do_:=TRUE;
	BULLS_EYE_GA.DoWhat:='unlock';
END_IF
END_ACTION

ACTION CHECK_STATE_active:
IF (PREWASH_WASH_POLICY.State='pre') THEN
	GVL.prewash:=TRUE;
	GVL.wash:=FALSE;
	GVL.rinse:=FALSE;
END_IF

IF (PREWASH_WASH_POLICY.State='rinse') THEN
	GVL.prewash:=FALSE;
	GVL.wash:=FALSE;
	GVL.rinse:=TRUE;
END_IF

IF (PREWASH_WASH_POLICY.State='wash') THEN
	GVL.prewash:=FALSE;
	GVL.wash:=TRUE;
	GVL.rinse:=FALSE;
END_IF

IF PREWASH_WASH_POLICY.State='fault' OR PREWASH_WASH_POLICY.State='end' THEN
	GVL.prewash:=FALSE;
	GVL.wash:=FALSE;
	GVL.rinse:=FALSE;
END_IF
END_ACTION

END_PROGRAM

// Device/Application/Visualization
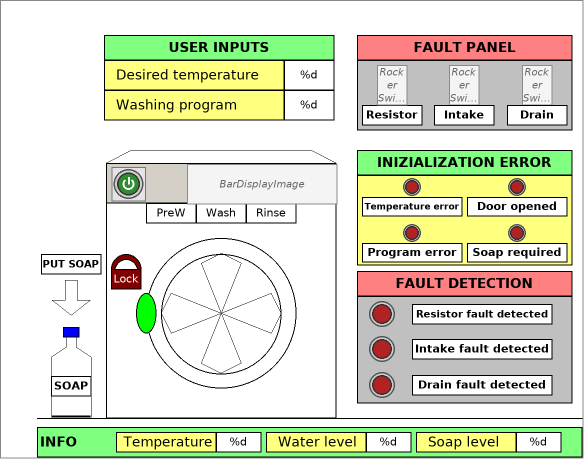
VISUALIZATION Visualization  // 584x459
    Line (37,418) (582,418)
    Rectangle (106,178 230x240)
    Ellipse (162,254 118x118)
    Rectangle (161,255 120x120)
        p1126004900: -GVL.waterlevel/3*2
    Ellipse (146,238 150x150)
    Ellipse (161,254 120x120)
    Polygon (221,253) (201,263) (221,313) (171,293) (161,313) (171,333) (221,313) (201,363) (221,373) (241,363) (221,313) (271,333) (281,313) (271,293) (221,313) (241,263)
        p2858320360: GVL.motor
    Ellipse (136,293 20x40), colour toggle: GVL.bulls_eye_open
        toggle GVL.bulls_eye_open
    Ellipse (111,254 30x30), colour toggle: GVL.bulls_eye_lock
    Ellipse (114,259 24x27)
    Rectangle (111,269 30x20), "Lock", colour toggle: GVL.bulls_eye_lock
    Rectangle (106,163 230x40)
    Rectangle (146,203 50x20), "PreW", colour toggle: GVL.prewash
    Rectangle (196,203 50x20), "Wash", colour toggle: GVL.wash
    Rectangle (246,203 50x20), "Rinse", colour toggle: GVL.rinse
    Polygon (106,163) (131,150) (311,150) (336,163)
    PowerSwitch (111,167 35x34), variable: GVL.run, behaviour: TOGGLE, style: Switch-PowerSwitch-Green
    BarDisplayImage (187,164 150x40), value: GVL.temperature, style: BarDisplayImage-Gray, scale format: %.0f, scale 0..90
    Polygon (51,417) (51,357) (66,347) (66,332) (76,332) (76,347) (91,357) (91,417)
    Rectangle (63,327 16x10)
    Rectangle (104,60 180x30), "Desired temperature"
        OnMouseDown: write GVL.temp_number via VisuDialogs.Numpad, min 0, max 100, format 0
    Rectangle (104,90 180x30), "Washing program"
        OnMouseDown: write GVL.prog_number via VisuDialogs.Numpad, min 0, max 100, format 0
    Rectangle (104,35 230x25), "USER INPUTS"
    Rectangle (284,60 50x30), "%d", text variable: GVL.temp_number
    Rectangle (284,90 50x30), "%d", text variable: GVL.prog_number
    Rectangle (37,427 545x30), "INFO"
    Rectangle (116,432 100x20), "Temperature"
    Rectangle (357,150 215x25), "INIZIALIZATION ERROR"
    Rectangle (216,432 45x20), "%d", text variable: GVL.temperature
    Rectangle (266,432 100x20), "Water level"
    Rectangle (366,432 45x20), "%d", text variable: GVL.waterlevel
    Rectangle (416,432 100x20), "Soap level"
    Rectangle (516,432 45x20), "%d", text variable: GVL.soaplevel
    Rectangle (357,175 215x90)
    Lamp1 (402,177 20x20), variable: GVL.temp_error, style: Lamp-Lamp1-Red
    Rectangle (362,197 100x19), "Temperature error"
    Lamp1 (507,177 20x20), variable: GVL.bulls_eye_open, style: Lamp-Lamp1-Red
    Rectangle (467,197 100x19), "Door opened"
    Lamp1 (402,223 20x20), variable: GVL.prog_error, style: Lamp-Lamp1-Red
    Rectangle (362,243 100x19), "Program error"
    Lamp1 (507,223 20x20), variable: GVL.soap_alarm, style: Lamp-Lamp1-Red
    Rectangle (467,243 100x19), "Soap required"
    Rectangle (357,35 215x25), "FAULT PANEL"
    Rectangle (357,60 215x70)
    Rectangle (362,105 60x20), "Resistor"
    RockerSwitch (377,65 30x40), variable: GVL.heat_fail, behaviour: TOGGLE, style: Switch-RockerSwitch-Red
    RockerSwitch (449,65 30x40), variable: GVL.water_in_fail, behaviour: TOGGLE, style: Switch-RockerSwitch-Red
    Rectangle (434,105 60x20), "Intake"
    RockerSwitch (522,65 30x40), variable: GVL.water_out_fail, behaviour: TOGGLE, style: Switch-RockerSwitch-Red
    Rectangle (507,105 60x20), "Drain"
    Rectangle (357,271 215x25), "FAULT DETECTION"
    Rectangle (357,296 215x107)
    Lamp1 (367,299 30x30), variable: GVL.heat_alarm, style: Lamp-Lamp1-Red
    Rectangle (412,304 140x20), "Resistor fault detected"
    Lamp1 (367,370 30x30), variable: GVL.water_out_alarm, style: Lamp-Lamp1-Red
    Lamp1 (367,334 30x30), variable: GVL.water_in_alarm, style: Lamp-Lamp1-Red
    Rectangle (412,339 140x20), "Intake fault detected"
    Rectangle (412,375 140x20), "Drain fault detected"
    Rectangle (52,416 38x0)
        p2773130477: -GVL.soaplevel
    Rectangle (51,376 40x20), "SOAP"
    Polygon (65,280) (65,300) (52,300) (71,315) (90,300) (77,300) (77,280), colour toggle: GVL.fillsoap
        toggle GVL.fillsoap
    Rectangle (41,254 60x20), "PUT SOAP"
END_VISUALIZATION
